INTERFACE I_ValueDeviationLimited

{attribute 'monitoring':='call'}
// Gets or sets the activation delay, before the deviation error is activated
PROPERTY ActivationDelay : TIME
GET
END_GET
SET
END_SET
END_PROPERTY

{attribute 'monitoring':='call'}
PROPERTY Enable : BOOL
GET
END_GET
SET
END_SET
END_PROPERTY

{attribute 'monitoring':='call'}
PROPERTY MaxDeviation : T_ControllerValue
GET
END_GET
SET
END_SET
END_PROPERTY

{attribute 'monitoring':='call'}
PROPERTY Status : E_ValueDeviationStatus
GET
END_GET
END_PROPERTY

END_INTERFACE

(* stored: Version 1.1.0.1, ProductVersion 3.1.4024.15
   Itf I_ValueDeviationLimited: Id {74d874eb-3985-0701-0aaa-9006c1ea4e23}
   Property ActivationDelay: Id {6cde609b-6483-0f7e-2418-a4e8988346c8}
   Get Get: Id {7b69c608-af78-0596-0ff3-b209aabc7e89}
   Set Set: Id {a9db1e01-6b0b-09ab-2dd9-c0d126ebcb9c}
   Property Enable: Id {cdd81f2e-f02d-0a1c-3a63-3d0f08203bf8}
   Get Get: Id {66d95846-6f4a-0ead-15f4-36825208aaf6}
   Set Set: Id {73a868f9-3377-0778-117c-1a15590ce107}
   Property MaxDeviation: Id {9fac01cf-ce34-0ab8-26d7-8ef175f4b975}
   Get Get: Id {2c56080e-1ecf-0f1a-14f2-ecd7cdc6128f}
   Set Set: Id {6bfcd3c6-8de1-03a4-0fd5-82145a7e0f77}
   Property Status: Id {60eb8bdb-398e-0a99-1c9b-5fa267ac1dfa}
   Get Get: Id {02ae5f25-93a9-0f78-3241-0b335bcf0312} *)
